FUNCTION_BLOCK INTERNAL FINAL FB_WriteRepeatedFieldFloatTests EXTENDS FB_TestSuite
VAR_INPUT
END_VAR
VAR_OUTPUT
END_VAR
VAR
    fbFieldCodec : FB_FieldCodecFloat;
END_VAR
(*
syntax = "proto3";

message MessageRepeatedFloat
{
  repeated float repeatedFloat = 4;
}


JSON:
{
  "repeatedFloat": [
    0, 1234.567, 1337.1337, -1.0, 12345678.321, 2147483647.65432
  ]
}

*)

ShouldWriteRepeatedFieldTheory();

METHOD PRIVATE ShouldWriteRepeatedField
VAR_IN_OUT CONSTANT
    aExpected   : ARRAY [*] OF BYTE;
END_VAR
VAR_INPUT
    aValues     : ARRAY [0..7] OF REAL;
    nLength     : UDINT;
    nTag        : UDINT;
    nBufferPosStart     : UDINT;
    nExpectedBufferPos  : UDINT;
    ipFieldCodec        : I_FieldCodec;
END_VAR
VAR_INST
    stState : ST_WriterInternalState;
END_VAR
VAR
    aActualBuffer       : ARRAY [0..63] OF BYTE;
    hr                  : HRESULT;

END_VAR
// Arrange
stState.nBufferPos := nBufferPosStart;
stState.nBufferSize := SIZEOF(aActualBuffer);

// Act
hr := F_WriteRepeatedField(aActualBuffer, stState, anyArray:= F_ToAnyType(aValues), anyFirstElem:= F_ToAnyType(aValues[0]), nLength, F_MakeTag(nTag, E_WireType.LengthDelimited), ipFieldCodec);

// Assert
AssertEquals_DINT(
    Expected:= S_OK,
    Actual:= hr,
    Message:= 'Expected S_OK instead of error');
    
{warning disable C0041}
AssertArrayEquals_BYTE(Expecteds:= aExpected, Actuals:= aActualBuffer, Message:= '');
 
AssertEquals_UDINT(
    Expected:= nExpectedBufferPos,
    Actual:= stState.nBufferPos,
    Message:= CONCAT('Expected stState.nBufferPos to equal ', TO_STRING(nExpectedBufferPos)));
END_METHOD

METHOD PRIVATE ShouldWriteRepeatedFieldTheory : REFERENCE TO FB_Test
VAR CONSTANT
    cRawValueZeroLength     : ARRAY[0..63] OF BYTE := [16#0A, 16#00];
    cRawValue1              : ARRAY[0..63] OF BYTE := [16#00, 16#22, 16#18, 16#00, 16#00, 16#00, 16#00, 16#25, 16#52, 16#9a, 16#44, 16#47, 16#24, 16#a7, 16#44, 16#00, 16#00, 16#80, 16#bf, 16#4e, 16#61, 16#3c, 16#4b, 16#00, 16#00, 16#00, 16#4f];  
END_VAR

VAR CONSTANT
    aExpectedZeroLength     : ARRAY [0..7] OF REAL := [0, 0, 0, 0, 0, 0, 0, 0];
    aExpected1              : ARRAY [0..7] OF REAL := [0, 1234.567, 1337.1337, -1.0, 12345678.321, 2147483647.65432];
END_VAR
TEST(__POUNAME());

ShouldWriteRepeatedField(aExpected:= cRawValueZeroLength, aValues:= aExpectedZeroLength, nLength:= 0, nTag:= 1, nBufferPosStart:= 0, nExpectedBufferPos:= 2, ipFieldCodec:= THIS^.fbFieldCodec);
ShouldWriteRepeatedField(aExpected:= cRawValue1, aValues:= aExpected1, nLength:= 6, nTag:= 4, nBufferPosStart:= 1, nExpectedBufferPos:= 27, ipFieldCodec:= THIS^.fbFieldCodec);

TEST_FINISHED_NAMED(__POUNAME());
END_METHOD

END_FUNCTION_BLOCK

(* stored: Version 1.1.0.1
   POU FB_WriteRepeatedFieldFloatTests: Id {240cd37b-8c50-4152-9ae3-4e86c180dbc9}, SpecialFunc None
   Method ShouldWriteRepeatedField: Id {556ca8ed-0648-4b96-8e11-0bb06b018aa5}
   Method ShouldWriteRepeatedFieldTheory: Id {73353956-3bc9-4eb0-9b4a-084cf1213422} *)
